Universal Robots PolyScope program: ProcessIntensity.urp

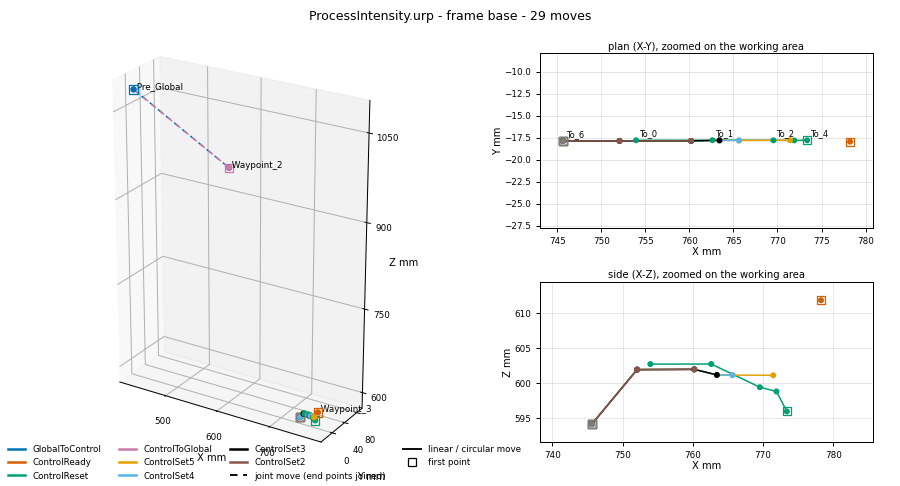
[picture p0: tool path of ProcessIntensity.urp in frame base, 29 of 46 moves have a stored position in this frame; points joined in program order, loops and branches not executed]
Program ProcessIntensity (installation=Youssef directory=/programs/Youssef createdIn=5.9.5.1031259 lastSavedIn=5.9.5.1031259 robotSerialNumber=20215500597)
Calibrated DH parameters: a=[0.000193, -0.066673, -0.391568, -0.000012, 0.00005, 0]; d=[0.162643, -472.05677, 465.132521, 7.058239, 0.099746, 0.099582]; alpha=[1.571116, 0.00089, 0.003862, 1.569269, -1.569248, 0]; deltaTheta=[0, -1.413394, 7.628392, 0.068187, 0, -0.000001]
Robot Program (runOnlyOnce=true)
  Call GlobalToControl
  Call ControlReady
  Call ControlReset
  Call ControlSet
  Call ControlStandby
  Call ControlToGlobal
SubProgram -> GlobalToControl
SubProgram -> ControlReady
SubProgram -> ControlReset
SubProgram -> ControlSet
SubProgram -> ControlSet1
SubProgram -> ControlSet2
SubProgram -> ControlSet3
SubProgram -> ControlSet4
SubProgram -> ControlSet5
SubProgram -> ControlStandby
SubProgram -> ControlToGlobal
SubProgram GlobalToControl (keepSynchronizedWithDisk=true) programFile=/programs/Youssef/GlobalToControl.urp
  MoveJ speed 60 deg/s, acceleration 80 deg/s^2 (useActiveTCP=true) feature=Base
    SafeHome (positionOptionType=SPEED_AND_ACCELERATION speed=1.047198 acceleration=1.396263 nextMotionTime=2)
    Waypoint Pre_Global: TCP in base x=424.817 y=-1.551 z=1080.554 mm, rx=-1.2067 ry=1.2116 rz=-1.2125 rad; joints [89.999, -90, 0, -89.996, -0.001, -0.002] deg; TCP offset x=0 y=0 z=191.5 mm, rx=0 ry=0 rz=0 rad
    URCap Gripper Activate (Robotiq_Grippers, Robotiq Inc.) dataModel(ResetAndActivateKey=false)
    URCap Gripper (Robotiq_Grippers, Robotiq Inc.) dataModel(position=100.0, force=0.0, speed=30.0, positionInDouble=100.0, forceInDouble=0.0, speedInDouble=30.0, slaveIds=[9], blocking=true)
    Waypoint Waypoint_2: TCP in base x=551.14 y=80.155 z=946.388 mm, rx=-1.3882 ry=1.5372 rz=-1.1084 rad; joints [175.158, -73.344, -0.017, -87.688, -91.199, -0.001] deg
    Waypoint Waypoint (Variable): variable(featureName=Control_Standby)
SubProgram ControlReady (keepSynchronizedWithDisk=true) programFile=/programs/Youssef/ControlReady.urp
  MoveJ speed 60 deg/s, acceleration 80 deg/s^2 (useActiveTCP=true) feature=Base
    Waypoint Waypoint (Variable): variable(featureName=Control_Standby)
    Waypoint Waypoint_3: TCP in base x=778.24 y=-17.942 z=611.823 mm, rx=-0.0636 ry=2.4704 rz=-0.2743 rad; joints [170.473, -63.159, 27.038, -93.122, -94.218, 75.99] deg
  MoveL speed 250 mm/s, acceleration 1200 mm/s^2 (useActiveTCP=true) feature=Base
    Waypoint Waypoint (Variable): variable(featureName=Control_R_End)
SubProgram ControlReset (keepSynchronizedWithDisk=true) programFile=/programs/Youssef/ControlReset.urp
  MoveL speed 250 mm/s, acceleration 1200 mm/s^2 (useActiveTCP=true) feature=Base
    Waypoint Waypoint (Variable): variable(featureName=Control_R_End)
    Waypoint To_4: motionParameters(jointSpeed=1.047198 jointAcceleration=1.396263 cartesianSpeed=0.1 cartesianAcceleration=1.2); TCP in base x=773.379 y=-17.782 z=595.99 mm, rx=-0.0637 ry=2.4704 rz=-0.2742 rad; joints [170.403, -66.53, 35.056, -97.772, -94.172, 75.95] deg
    Waypoint To_3: motionParameters(jointSpeed=1.047198 jointAcceleration=1.396263 cartesianSpeed=0.1 cartesianAcceleration=1.2); TCP in base x=771.893 y=-17.795 z=598.835 mm, rx=-0.0637 ry=2.4705 rz=-0.2742 rad; joints [170.378, -66.476, 34.483, -97.248, -94.158, 75.93] deg
    Waypoint To_2: motionParameters(jointSpeed=1.047198 jointAcceleration=1.396263 cartesianSpeed=0.1 cartesianAcceleration=1.2); TCP in base x=769.54 y=-17.783 z=599.437 mm, rx=-0.0638 ry=2.4705 rz=-0.2742 rad; joints [170.339, -66.884, 34.994, -97.353, -94.131, 75.897] deg
    Waypoint To_1: motionParameters(jointSpeed=1.047198 jointAcceleration=1.396263 cartesianSpeed=0.1 cartesianAcceleration=1.2); TCP in base x=762.609 y=-17.768 z=602.737 mm, rx=-0.0638 ry=2.4705 rz=-0.2742 rad; joints [170.223, -67.881, 35.915, -97.286, -94.059, 75.807] deg
    Waypoint To_0: motionParameters(jointSpeed=1.047198 jointAcceleration=1.396263 cartesianSpeed=0.1 cartesianAcceleration=1.2); TCP in base x=753.941 y=-17.776 z=602.724 mm, rx=-0.0637 ry=2.4705 rz=-0.2742 rad; joints [170.071, -69.568, 38.384, -98.074, -93.963, 75.694] deg
    Waypoint Waypoint (Variable): variable(featureName=Control_Standby)
SubProgram ControlSet (keepSynchronizedWithDisk=false) programFile=/programs/Youssef/ControlSet.urp
  If GP_int_in[6]≟5
    Call ControlSet5
  ElseIf GP_int_in[6]≟4
    Call ControlSet4
  ElseIf GP_int_in[6]≟3
    Call ControlSet3
  ElseIf GP_int_in[6]≟2
    Call ControlSet2
  Else 
    Call ControlSet1
SubProgram ControlStandby (keepSynchronizedWithDisk=true) programFile=/programs/Youssef/ControlStandby.urp
  MoveJ speed 60 deg/s, acceleration 80 deg/s^2 (useActiveTCP=true) feature=Base
    Waypoint Waypoint (Variable): variable(featureName=Control_Standby)
SubProgram ControlToGlobal (keepSynchronizedWithDisk=true) programFile=/programs/Youssef/ControlToGlobal.urp
  MoveJ speed 60 deg/s, acceleration 80 deg/s^2 (useActiveTCP=true) feature=Base
    Waypoint Waypoint (Variable): variable(featureName=Control_Standby)
    Waypoint Waypoint_11: TCP in base x=551.14 y=80.155 z=946.388 mm, rx=-1.3882 ry=1.5372 rz=-1.1084 rad; joints [175.158, -73.344, -0.017, -87.688, -91.199, -0.001] deg
    URCap Gripper (Robotiq_Grippers, Robotiq Inc.) dataModel(position=0.0, force=0.0, speed=30.0, positionInDouble=0.0, forceInDouble=0.0, speedInDouble=30.0, slaveIds=[9], blocking=true)
    URCap Gripper Activate (Robotiq_Grippers, Robotiq Inc.) dataModel(ResetAndActivateKey=false)
    Waypoint Pre_Global_1: TCP in base x=424.817 y=-1.551 z=1080.554 mm, rx=-1.2067 ry=1.2116 rz=-1.2125 rad; joints [89.999, -90, 0, -89.996, -0.001, -0.002] deg
    SafeHome (positionOptionType=SPEED_AND_ACCELERATION speed=1.047198 acceleration=1.396263 nextMotionTime=2)
SubProgram ControlSet5 (keepSynchronizedWithDisk=false) programFile=/programs/Youssef/ControlSet5.urp
  MoveL speed 250 mm/s, acceleration 1200 mm/s^2 (useActiveTCP=true) feature=Base
    Waypoint Waypoint (Variable): variable(featureName=Control_Standby)
    Waypoint Waypoint (Variable): variable(featureName=Control_R_Strt)
    Waypoint To_6: TCP in base x=745.639 y=-17.849 z=594.209 mm, rx=-0.0636 ry=2.4703 rz=-0.2743 rad; joints [169.914, -71.977, 43.233, -100.537, -93.87, 75.587] deg
  MoveL speed 250 mm/s, acceleration 1200 mm/s^2 (useActiveTCP=true) feature=Base
    Waypoint Adjust_2: TCP in base x=752.062 y=-17.854 z=601.945 mm, rx=-0.0636 ry=2.4704 rz=-0.2743 rad; joints [170.031, -70.021, 39.176, -98.427, -93.941, 75.669] deg
    Waypoint To_7: TCP in base x=760.195 y=-17.853 z=601.978 mm, rx=-0.0636 ry=2.4703 rz=-0.2743 rad; joints [170.175, -68.462, 36.913, -97.718, -94.032, 75.776] deg
  MoveL speed 250 mm/s, acceleration 1200 mm/s^2 (useActiveTCP=true) feature=Base
    Waypoint To_8: TCP in base x=763.415 y=-17.79 z=601.185 mm, rx=-0.0639 ry=2.4729 rz=-0.2738 rad; joints [170.234, -67.759, 35.895, -97.252, -94.064, 75.817] deg
  MoveL speed 250 mm/s, acceleration 1200 mm/s^2 (useActiveTCP=true) feature=Base
    Waypoint To_9: TCP in base x=765.628 y=-17.8 z=601.16 mm, rx=-0.0639 ry=2.4729 rz=-0.2738 rad; joints [170.271, -67.314, 35.235, -97.032, -94.088, 75.845] deg
  MoveL speed 250 mm/s, acceleration 1200 mm/s^2 (useActiveTCP=true) feature=Base
    Waypoint To_5: TCP in base x=771.437 y=-17.779 z=601.135 mm, rx=-0.064 ry=2.473 rz=-0.2737 rad; joints [170.371, -66.115, 33.43, -96.418, -94.148, 75.918] deg
SubProgram ControlSet4 (keepSynchronizedWithDisk=false) programFile=/programs/Youssef/ControlSet4.urp
  MoveL speed 250 mm/s, acceleration 1200 mm/s^2 (useActiveTCP=true) feature=Base
    Waypoint Waypoint (Variable): variable(featureName=Control_Standby)
    Waypoint Waypoint (Variable): variable(featureName=Control_R_Strt)
    Waypoint To_13: TCP in base x=745.639 y=-17.849 z=594.209 mm, rx=-0.0636 ry=2.4703 rz=-0.2743 rad; joints [169.914, -71.977, 43.233, -100.537, -93.87, 75.587] deg
  MoveL speed 250 mm/s, acceleration 1200 mm/s^2 (useActiveTCP=true) feature=Base
    Waypoint Adjust_3: TCP in base x=752.062 y=-17.854 z=601.945 mm, rx=-0.0636 ry=2.4704 rz=-0.2743 rad; joints [170.031, -70.021, 39.176, -98.427, -93.941, 75.669] deg
    Waypoint To_14: TCP in base x=760.195 y=-17.853 z=601.978 mm, rx=-0.0636 ry=2.4703 rz=-0.2743 rad; joints [170.175, -68.462, 36.913, -97.718, -94.032, 75.776] deg
  MoveL speed 250 mm/s, acceleration 1200 mm/s^2 (useActiveTCP=true) feature=Base
    Waypoint To_15: TCP in base x=763.415 y=-17.79 z=601.185 mm, rx=-0.0639 ry=2.4729 rz=-0.2738 rad; joints [170.234, -67.759, 35.895, -97.252, -94.064, 75.817] deg
  MoveL speed 250 mm/s, acceleration 1200 mm/s^2 (useActiveTCP=true) feature=Base
    Waypoint To_16: TCP in base x=765.628 y=-17.8 z=601.16 mm, rx=-0.0639 ry=2.4729 rz=-0.2738 rad; joints [170.271, -67.314, 35.235, -97.032, -94.088, 75.845] deg
SubProgram ControlSet3 (keepSynchronizedWithDisk=false) programFile=/programs/Youssef/ControlSet3.urp
  MoveL speed 250 mm/s, acceleration 1200 mm/s^2 (useActiveTCP=true) feature=Base
    Waypoint Waypoint (Variable): variable(featureName=Control_Standby)
    Waypoint Waypoint (Variable): variable(featureName=Control_R_Strt)
    Waypoint To_10: TCP in base x=745.639 y=-17.849 z=594.209 mm, rx=-0.0636 ry=2.4703 rz=-0.2743 rad; joints [169.914, -71.977, 43.233, -100.537, -93.87, 75.587] deg
  MoveL speed 250 mm/s, acceleration 1200 mm/s^2 (useActiveTCP=true) feature=Base
    Waypoint Adjust_1: TCP in base x=752.062 y=-17.854 z=601.945 mm, rx=-0.0636 ry=2.4704 rz=-0.2743 rad; joints [170.031, -70.021, 39.176, -98.427, -93.941, 75.669] deg
    Waypoint To_11: TCP in base x=760.195 y=-17.853 z=601.978 mm, rx=-0.0636 ry=2.4703 rz=-0.2743 rad; joints [170.175, -68.462, 36.913, -97.718, -94.032, 75.776] deg
  MoveL speed 250 mm/s, acceleration 1200 mm/s^2 (useActiveTCP=true) feature=Base
    Waypoint To_12: TCP in base x=763.415 y=-17.79 z=601.185 mm, rx=-0.0639 ry=2.4729 rz=-0.2738 rad; joints [170.234, -67.759, 35.895, -97.252, -94.064, 75.817] deg
SubProgram ControlSet2 (keepSynchronizedWithDisk=false) programFile=/programs/Youssef/ControlSet2.urp
  MoveL speed 250 mm/s, acceleration 1200 mm/s^2 (useActiveTCP=true) feature=Base
    Waypoint Waypoint (Variable): variable(featureName=Control_Standby)
    Waypoint Waypoint (Variable): variable(featureName=Control_R_Strt)
    Waypoint To_17: TCP in base x=745.639 y=-17.849 z=594.209 mm, rx=-0.0636 ry=2.4703 rz=-0.2743 rad; joints [169.914, -71.977, 43.233, -100.537, -93.87, 75.587] deg
  MoveL speed 250 mm/s, acceleration 1200 mm/s^2 (useActiveTCP=true) feature=Base
    Waypoint Adjust_4: TCP in base x=752.062 y=-17.854 z=601.945 mm, rx=-0.0636 ry=2.4704 rz=-0.2743 rad; joints [170.031, -70.021, 39.176, -98.427, -93.941, 75.669] deg
    Waypoint To_18: TCP in base x=760.195 y=-17.853 z=601.978 mm, rx=-0.0636 ry=2.4703 rz=-0.2743 rad; joints [170.175, -68.462, 36.913, -97.718, -94.032, 75.776] deg
SubProgram ControlSet1 (keepSynchronizedWithDisk=false) programFile=/programs/Youssef/ControlSet1.urp
  MoveL speed 250 mm/s, acceleration 1200 mm/s^2 (useActiveTCP=true) feature=Base
    Waypoint Waypoint (Variable): variable(featureName=Control_Standby)
    Waypoint Waypoint (Variable): variable(featureName=Control_R_Strt)
    Waypoint To_19: TCP in base x=745.639 y=-17.849 z=594.209 mm, rx=-0.0636 ry=2.4703 rz=-0.2743 rad; joints [169.914, -71.977, 43.233, -100.537, -93.87, 75.587] deg
